TYPE csp_transfer_upstacker_carton_backstop_status :
(
	NONE							:= 0,
	PRESENT							:= 1,
	ABSENT							:= 2	
);
END_TYPE

(* stored: Version 1.1.0.1, ProductVersion 3.1.4022.12
   DUT csp_transfer_upstacker_carton_backstop_status: Id {da568289-173b-4404-b6a6-b679d21af68c} *)
